Staubli VAL3: CheckCellFormat.pgx

program CheckCellFormat(string& x_sCellNumber[], bool& x_bMatchOK[])
  local num l_i
  local bool l_bDigitOK
  local string l_sWrkString
begin
  // this routines checks if the format of the string used to point on a cell
  // of the cognex speadsheet matches the format of native command
  //
  // Input Param
  //  x_sCellNumber  : Cell number in string format. Must be :
  //            First digit is a letter (A-Z) for Column number
  //            3 next digits is a number for Row number
  //
  // Output Param
  //  x_bMatchOK  : TRUE if format of the String passed as parameter is OK
  //------------------------------------------------------------
  x_bMatchOK=true
  if len(x_sCellNumber)>=2
    // first digit must be in range 'A-Z' or 'a-z'
    call checkColValue(mid(x_sCellNumber,1,0),l_bDigitOK)
    if l_bDigitOK
      l_sWrkString=right(x_sCellNumber,len(x_sCellNumber)-1)
      for l_i=1 to len(l_sWrkString)
        l_bDigitOK=l_bDigitOK and (asc(mid(l_sWrkString,l_i,0),0)>=(asc("0",0))) and (asc(mid(l_sWrkString,l_i,0),0)<=(asc("9",0)))
      endFor
      if l_bDigitOK
        l_sWrkString=mid("000",3-len(l_sWrkString),0)+l_sWrkString
      endIf
      x_sCellNumber=mid(x_sCellNumber,1,0)+l_sWrkString
    else
      x_bMatchOK=false
    endIf
  else
    x_bMatchOK=false
  endIf
end
